Fanuc TP program (LS listing): VACUUM_ON.LS

/PROG  VACUUM_ON	  Macro
/ATTR
OWNER		= MNEDITOR;
COMMENT		= "Vacuum On";
PROG_SIZE	= 230;
CREATE		= DATE 25-09-17  TIME 15:38:02;
MODIFIED	= DATE 25-09-17  TIME 15:38:02;
FILE_NAME	= T_VACON;
VERSION		= 0;
LINE_COUNT	= 4;
MEMORY_SIZE	= 586;
PROTECT		= READ_WRITE;
STORAGE		= SHADOW;
TCD:  STACK_SIZE	= 0,
      TASK_PRIORITY	= 50,
      TIME_SLICE	= 0,
      BUSY_LAMP_OFF	= 0,
      ABORT_REQUEST	= 0,
      PAUSE_REQUEST	= 0;
DEFAULT_GROUP	= *,*,*,*,*;
CONTROL_CODE	= 00000000 00000000;
LOCAL_REGISTERS	= 0,0,0;
/APPL
/MN
   1:  --dn:pgri[9] ;
   2:  RO[1]=OFF ;
   3:  RO[2]=ON ;
   4:  WAIT    .25(sec) ;
/POS
/END
